Fanuc KAREL source: kb00160.KL

-- PROVISIONAL review KL for V770-1; original PC SHA256 35c2c6960d5f7ffd00b2fc5eca39d759b1822c00960d404919fa5b8f00fcf4b6
-- Incomplete behavior may be omitted. Consult companion uncertainty JSON. Do not deploy.
PROGRAM KB00160
%NOLOCKGROUP
BEGIN
  -- UNRESOLVED_PC offsets 5-12; opcodes 9D,23
  -- UNRESOLVED_PC offsets 17-24; opcodes 9D,23
  -- UNRESOLVED_PC offsets 29-36; opcodes 9D,23
  -- UNRESOLVED_PC offsets 41-69; opcodes 27,22,22,22,22,31
  -- UNRESOLVED_PC offsets 74-78; opcodes 7F
END KB00160
